// TIA Portal V20 program export: 0 tag tables, 0 data types, 1 data blocks, 3 code blocks (in call order from the OBs), 2 instance data blocks

DATA_BLOCK "MotorSequence_Settings"   // DB2
{ S7_Optimized_Access := 'FALSE' }
VERSION : 1.0
// stored: AutoNumber true, DBAccessibleFromOPCUA true, DBAccessibleFromWebserver true, IsOnlyStoredInLoadMemory false, IsWriteProtectedInAS false
   VAR RETAIN
      StartInterval : Time := T#2S;
      StopInterval : Time := T#2S;
   END_VAR
BEGIN
END_DATA_BLOCK

ORGANIZATION_BLOCK "Main"   // OB1, LAD, ProgramCycle
TITLE = "Main Program Sweep (Cycle)"
{ S7_Optimized_Access := 'TRUE' }
VERSION : 0.1
// stored: AutoNumber false, IsIECCheckEnabled false, SetENOAutomatically false
   VAR_INPUT
      Initial_Call : Bool;
      Remanence : Bool;
   END_VAR
BEGIN

REGION Network 1
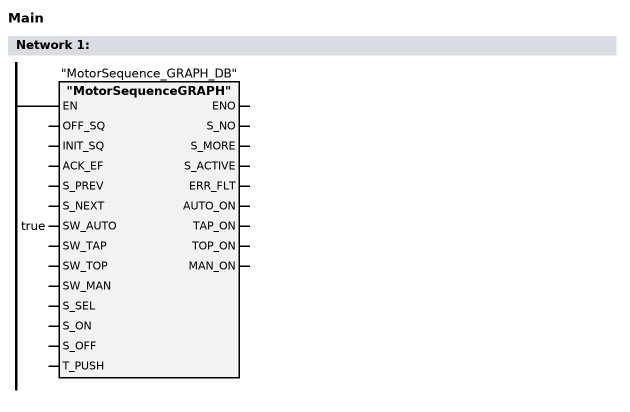
   RUNG wire#powerrail
      "MotorSequence_GRAPH_DB"(SW_AUTO := true, OFF_SQ :=, INIT_SQ :=, ACK_EF :=, S_PREV :=, S_NEXT :=, SW_TAP :=, SW_TOP :=, SW_MAN :=, S_SEL :=, S_ON :=, S_OFF :=, T_PUSH :=, S_NO =>, S_MORE =>, S_ACTIVE =>, ERR_FLT =>, AUTO_ON =>, TAP_ON =>, TOP_ON =>, MAN_ON =>)
   END_RUNG
   // the same network as SCL:
   "MotorSequence_GRAPH_DB"(SW_AUTO := true);   // "MotorSequenceGRAPH"
END_REGION
END_ORGANIZATION_BLOCK

FUNCTION_BLOCK "MotorSequenceGRAPH"   // FB2, GRAPH
VERSION : 0.1
// stored: AcknowledgeErrorsRequired true, AutoNumber false, GraphVersion 6.0, InitialValuesAcquisition false, IsIECCheckEnabled false, LanguageInNetworks LAD, LockOperatingMode false, PermanentILProcessingInMANMode false, SetENOAutomatically false, SkipSteps false, UDAEnableTagReadback false, WithAlarmHandling true
   // inherited from GRAPH_BASE
   VAR
      OFF_SQ_BASE : Bool;
   END_VAR
   VAR_INPUT
      OFF_SQ { ExternalAccessible := 'False'; ExternalVisible := 'False'; ExternalWritable := 'False'} : Bool := false;   // 关闭顺控器
      INIT_SQ { ExternalAccessible := 'False'; ExternalVisible := 'False'; ExternalWritable := 'False'} : Bool := false;   // 将顺序设置为初始状态
      ACK_EF { ExternalAccessible := 'False'; ExternalVisible := 'False'; ExternalWritable := 'False'} : Bool := false;   // 确认所有的错误和故障
      S_PREV { ExternalAccessible := 'False'; ExternalVisible := 'False'; ExternalWritable := 'False'} : Bool := false;   // 在S_NO输出参数中显示前导步
      S_NEXT { ExternalAccessible := 'False'; ExternalVisible := 'False'; ExternalWritable := 'False'} : Bool := false;   // 在S_NO输出参数中显示后续步。
      SW_AUTO { ExternalAccessible := 'False'; ExternalVisible := 'False'; ExternalWritable := 'False'} : Bool := false;   // 自动模式
      SW_TAP { ExternalAccessible := 'False'; ExternalVisible := 'False'; ExternalWritable := 'False'} : Bool := false;   // 半自动/转换条件切换
      SW_TOP { ExternalAccessible := 'False'; ExternalVisible := 'False'; ExternalWritable := 'False'} : Bool := false;   // 半自动/忽略转换条件
      SW_MAN { ExternalAccessible := 'False'; ExternalVisible := 'False'; ExternalWritable := 'False'} : Bool := false;   // 手动模式
      S_SEL { ExternalAccessible := 'False'; ExternalVisible := 'False'; ExternalWritable := 'False'} : Int := 0;   // 选择要在 S_NO中输出的步。
      S_ON { ExternalAccessible := 'False'; ExternalVisible := 'False'; ExternalWritable := 'False'} : Bool := false;   // 激活S_NO 中显示的步。
      S_OFF { ExternalAccessible := 'False'; ExternalVisible := 'False'; ExternalWritable := 'False'} : Bool := false;   // 禁用 S_NO 中标识的步
      T_PUSH { ExternalAccessible := 'False'; ExternalVisible := 'False'; ExternalWritable := 'False'} : Bool := false;   // 允许在半自动模式下跳过转换条件。
   END_VAR
   VAR_OUTPUT
      S_NO { ExternalAccessible := 'False'; ExternalVisible := 'False'; ExternalWritable := 'False'} : Int := 0;   // 步编号
      S_MORE { ExternalAccessible := 'False'; ExternalVisible := 'False'; ExternalWritable := 'False'} : Bool := false;   // 更多步可用，并可在S_NO中显示。
      S_ACTIVE { ExternalAccessible := 'False'; ExternalVisible := 'False'; ExternalWritable := 'False'} : Bool := false;   // 在S_NO 中显示的步是激活的。
      ERR_FLT { ExternalAccessible := 'False'; ExternalVisible := 'False'; ExternalWritable := 'False'} : Bool := false;   // 互锁条件或监控条件组出错
      AUTO_ON { ExternalAccessible := 'False'; ExternalVisible := 'False'; ExternalWritable := 'False'} : Bool := false;   // 当前为自动模式
      TAP_ON { ExternalAccessible := 'False'; ExternalVisible := 'False'; ExternalWritable := 'False'} : Bool := false;   // 已启用SW_TAP模式。
      TOP_ON { ExternalAccessible := 'False'; ExternalVisible := 'False'; ExternalWritable := 'False'} : Bool := false;   // 启用半自动模式/忽略转换条件。
      MAN_ON { ExternalAccessible := 'False'; ExternalVisible := 'False'; ExternalWritable := 'False'} : Bool := false;   // 已启用手动模式。
   END_VAR
BEGIN
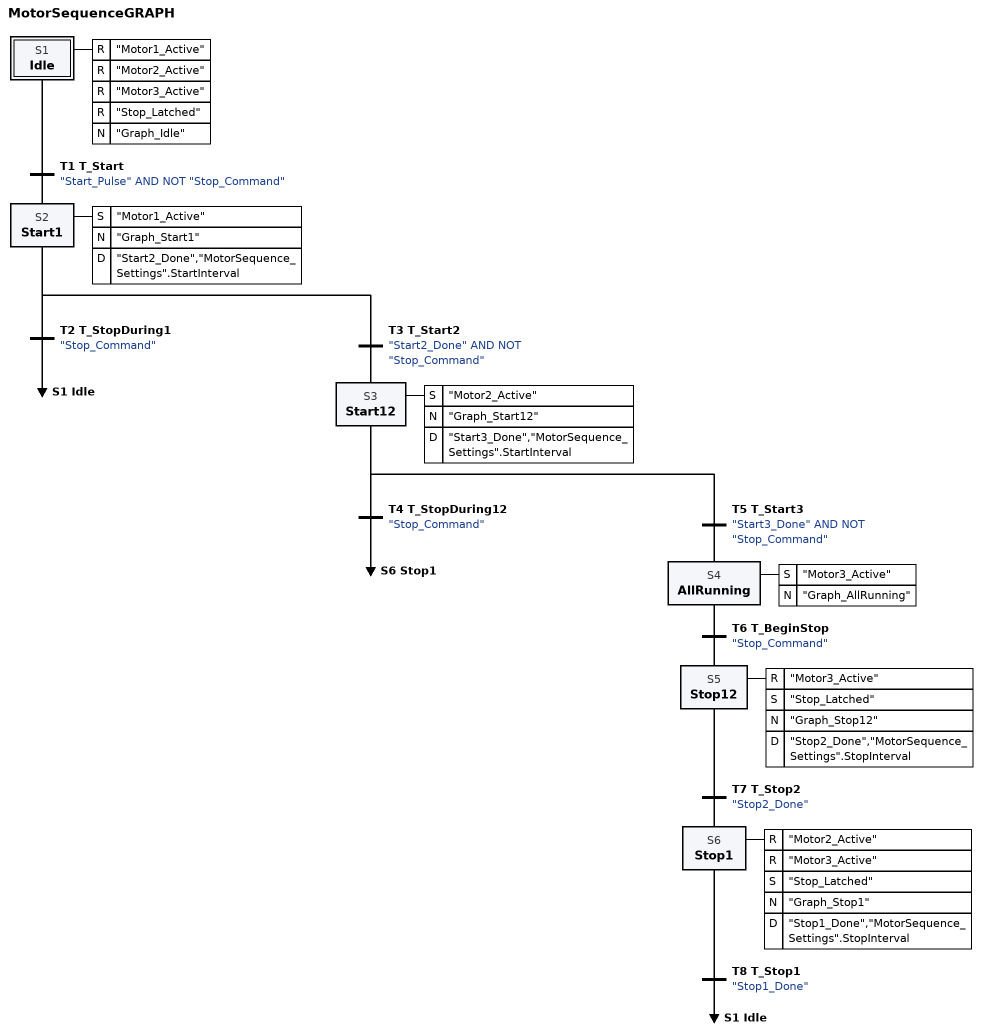
   // permanent pre-instructions
   NETWORK 1
      "Start_Pulse" := "Start_Command" AND NOT "Start_Previous";

   // sequencer 1: 三电机顺序启停：DB2可设间隔
   // 停止优先；停止阶段保持到全部停止；长按启动不自动重启。使用GRAPH原生D延时动作。
   INITIAL_STEP Idle:   // S1, max time T#0ms, warning time T#0ms
      supervision V := "Stop_Command" AND NOT "Stop_Command";
      // 空闲：全部停止，等待新的启动上升沿
              R    "Motor1_Active"
              R    "Motor2_Active"
              R    "Motor3_Active"
              R    "Stop_Latched"
              N    "Graph_Idle"
   END_STEP
   TRANSITION T_Start FROM Idle TO Start1   // T1
      := "Start_Pulse" AND NOT "Stop_Command";
   END_TRANSITION
   STEP Start1:   // S2, max time T#0ms, warning time T#0ms
      supervision V := "Stop_Command" AND NOT "Stop_Command";
      // 1号运行：等待启动间隔，停止优先
              S    "Motor1_Active"
              N    "Graph_Start1"
              D    "Start2_Done","MotorSequence_Settings".StartInterval
   END_STEP
   TRANSITION T_StopDuring1 FROM Start1 TO Idle   // T2, jump
      := "Stop_Command";
   END_TRANSITION
   TRANSITION T_Start2 FROM Start1 TO Start12   // T3
      := "Start2_Done" AND NOT "Stop_Command";
   END_TRANSITION
   STEP Start12:   // S3, max time T#0ms, warning time T#0ms
      supervision V := "Stop_Command" AND NOT "Stop_Command";
      // 1、2号运行：等待启动间隔，停止可跳至只留1号
              S    "Motor2_Active"
              N    "Graph_Start12"
              D    "Start3_Done","MotorSequence_Settings".StartInterval
   END_STEP
   TRANSITION T_StopDuring12 FROM Start12 TO Stop1   // T4, jump
      := "Stop_Command";
   END_TRANSITION
   TRANSITION T_Start3 FROM Start12 TO AllRunning   // T5
      := "Start3_Done" AND NOT "Stop_Command";
   END_TRANSITION
   STEP AllRunning:   // S4, max time T#0ms, warning time T#0ms
      supervision V := "Stop_Command" AND NOT "Stop_Command";
      // 三台电机全部运行，等待停止
              S    "Motor3_Active"
              N    "Graph_AllRunning"
   END_STEP
   TRANSITION T_BeginStop FROM AllRunning TO Stop12   // T6
      := "Stop_Command";
   END_TRANSITION
   STEP Stop12:   // S5, max time T#0ms, warning time T#0ms
      supervision V := "Stop_Command" AND NOT "Stop_Command";
      // 立即停3号，锁存停止序列，等待停止间隔
              R    "Motor3_Active"
              S    "Stop_Latched"
              N    "Graph_Stop12"
              D    "Stop2_Done","MotorSequence_Settings".StopInterval
   END_STEP
   TRANSITION T_Stop2 FROM Stop12 TO Stop1   // T7
      := "Stop2_Done";
   END_TRANSITION
   STEP Stop1:   // S6, max time T#0ms, warning time T#0ms
      supervision V := "Stop_Command" AND NOT "Stop_Command";
      // 立即停2号，保持1号至停止间隔结束
              R    "Motor2_Active"
              R    "Motor3_Active"
              S    "Stop_Latched"
              N    "Graph_Stop1"
              D    "Stop1_Done","MotorSequence_Settings".StopInterval
   END_STEP
   TRANSITION T_Stop1 FROM Stop1 TO Idle   // T8, jump
      := "Stop1_Done";
   END_TRANSITION

   // permanent post-instructions
   NETWORK 1
      "Motor_1" := "Motor1_Active";
   NETWORK 2
      "Motor_2" := "Motor2_Active";
   NETWORK 3
      "Motor_3" := "Motor3_Active";
   NETWORK 4
      "Start_Previous" := "Start_Command";
END_FUNCTION_BLOCK

FUNCTION_BLOCK "MotorSequenceLAD"   // FB1, LAD
{ S7_Optimized_Access := 'TRUE' }
VERSION : 0.1
// stored: AutoNumber true, IsIECCheckEnabled false, IsRetainMemResEnabled false, MemoryReserve 100, SetENOAutomatically false, UDAEnableTagReadback false
   VAR
      Start2 { S7_SetPoint := 'True'} : TON_TIME;
      Start3 { S7_SetPoint := 'True'} : TON_TIME;
      Stop2 { S7_SetPoint := 'True'} : TON_TIME;
      Stop1 { S7_SetPoint := 'True'} : TON_TIME;
   END_VAR
BEGIN

REGION Network 1: 启动上升沿，仅接受新的按钮动作
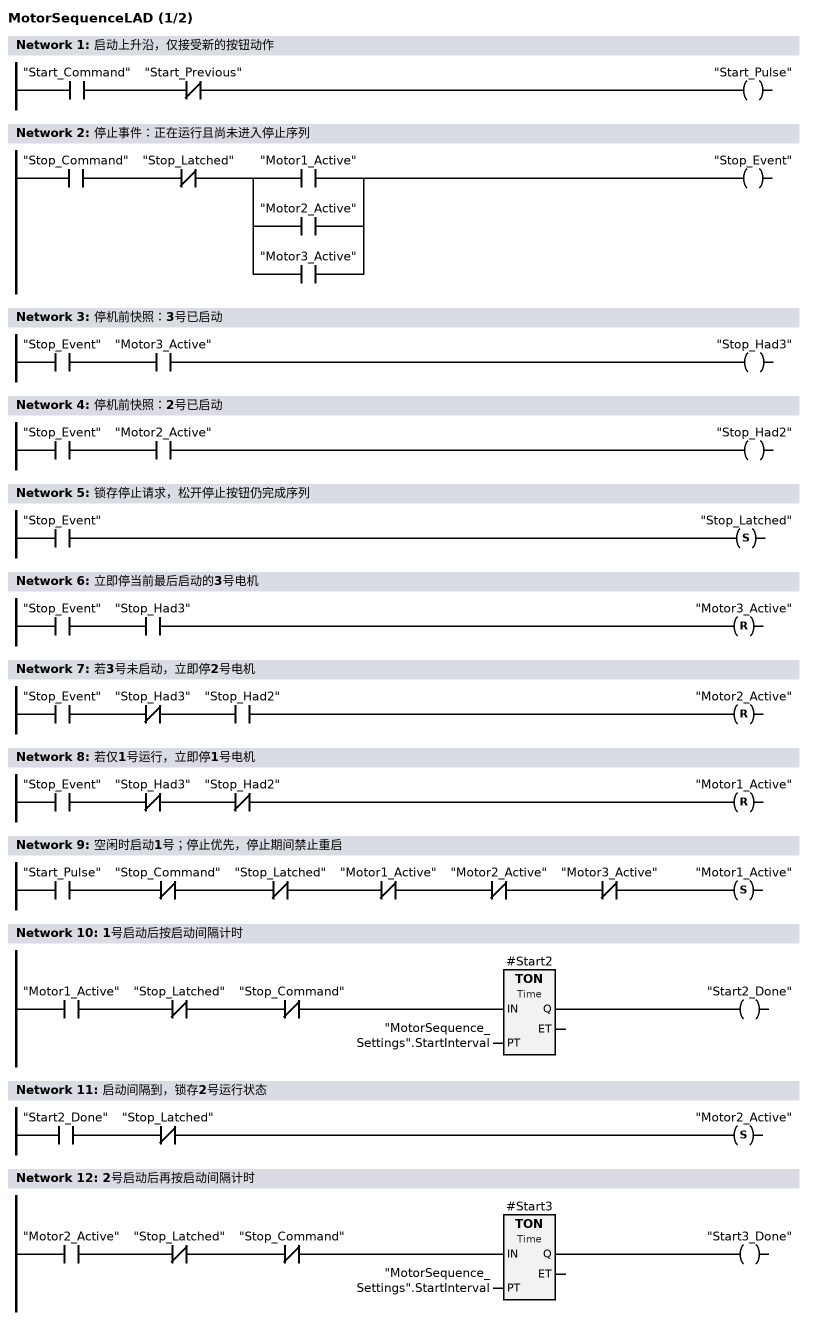
   RUNG wire#powerrail
      Contact( "Start_Command" )
      I_Contact( "Start_Previous" )
      Coil( "Start_Pulse" )
   END_RUNG
   // the same network as SCL:
   "Start_Pulse" := "Start_Command" AND NOT "Start_Previous";
END_REGION

REGION Network 2: 停止事件：正在运行且尚未进入停止序列
   RUNG wire#powerrail
      Contact( "Stop_Command" )
      I_Contact( "Stop_Latched" )
      wire#w1
      Contact( "Motor1_Active" )
      wire#w2
      Coil( "Stop_Event" )
   END_RUNG
   RUNG wire#w1
      Contact( "Motor2_Active" )
   END_RUNG wire#w2
   RUNG wire#w1
      Contact( "Motor3_Active" )
   END_RUNG wire#w2
   // the same network as SCL:
   "Stop_Event" := "Stop_Command" AND NOT "Stop_Latched" AND ("Motor1_Active" OR "Motor2_Active" OR "Motor3_Active");
END_REGION

REGION Network 3: 停机前快照：3号已启动
   RUNG wire#powerrail
      Contact( "Stop_Event" )
      Contact( "Motor3_Active" )
      Coil( "Stop_Had3" )
   END_RUNG
   // the same network as SCL:
   "Stop_Had3" := "Stop_Event" AND "Motor3_Active";
END_REGION

REGION Network 4: 停机前快照：2号已启动
   RUNG wire#powerrail
      Contact( "Stop_Event" )
      Contact( "Motor2_Active" )
      Coil( "Stop_Had2" )
   END_RUNG
   // the same network as SCL:
   "Stop_Had2" := "Stop_Event" AND "Motor2_Active";
END_REGION

REGION Network 5: 锁存停止请求，松开停止按钮仍完成序列
   RUNG wire#powerrail
      Contact( "Stop_Event" )
      S_Coil( "Stop_Latched" )
   END_RUNG
   // the same network as SCL:
   IF "Stop_Event" THEN "Stop_Latched" := TRUE; END_IF;
END_REGION

REGION Network 6: 立即停当前最后启动的3号电机
   RUNG wire#powerrail
      Contact( "Stop_Event" )
      Contact( "Stop_Had3" )
      R_Coil( "Motor3_Active" )
   END_RUNG
   // the same network as SCL:
   IF "Stop_Event" AND "Stop_Had3" THEN "Motor3_Active" := FALSE; END_IF;
END_REGION

REGION Network 7: 若3号未启动，立即停2号电机
   RUNG wire#powerrail
      Contact( "Stop_Event" )
      I_Contact( "Stop_Had3" )
      Contact( "Stop_Had2" )
      R_Coil( "Motor2_Active" )
   END_RUNG
   // the same network as SCL:
   IF "Stop_Event" AND NOT "Stop_Had3" AND "Stop_Had2" THEN "Motor2_Active" := FALSE; END_IF;
END_REGION

REGION Network 8: 若仅1号运行，立即停1号电机
   RUNG wire#powerrail
      Contact( "Stop_Event" )
      I_Contact( "Stop_Had3" )
      I_Contact( "Stop_Had2" )
      R_Coil( "Motor1_Active" )
   END_RUNG
   // the same network as SCL:
   IF "Stop_Event" AND NOT "Stop_Had3" AND NOT "Stop_Had2" THEN "Motor1_Active" := FALSE; END_IF;
END_REGION

REGION Network 9: 空闲时启动1号；停止优先，停止期间禁止重启
   RUNG wire#powerrail
      Contact( "Start_Pulse" )
      I_Contact( "Stop_Command" )
      I_Contact( "Stop_Latched" )
      I_Contact( "Motor1_Active" )
      I_Contact( "Motor2_Active" )
      I_Contact( "Motor3_Active" )
      S_Coil( "Motor1_Active" )
   END_RUNG
   // the same network as SCL:
   IF "Start_Pulse" AND NOT "Stop_Command" AND NOT "Stop_Latched" AND NOT "Motor1_Active" AND NOT "Motor2_Active" AND NOT "Motor3_Active" THEN
       "Motor1_Active" := TRUE;
   END_IF;
END_REGION

REGION Network 10: 1号启动后按启动间隔计时
   RUNG wire#powerrail
      Contact( "Motor1_Active" )
      I_Contact( "Stop_Latched" )
      I_Contact( "Stop_Command" )
      { S7_Templates := "time_type := Time" } #Start2.TON(pt := "MotorSequence_Settings".StartInterval, et =>)
      Coil( "Start2_Done" )
   END_RUNG
   // the same network as SCL:
   #Start2(IN := "Motor1_Active" AND NOT "Stop_Latched" AND NOT "Stop_Command",   // TON
           PT := "MotorSequence_Settings".StartInterval);
   "Start2_Done" := #Start2.Q;
END_REGION

REGION Network 11: 启动间隔到，锁存2号运行状态
   RUNG wire#powerrail
      Contact( "Start2_Done" )
      I_Contact( "Stop_Latched" )
      S_Coil( "Motor2_Active" )
   END_RUNG
   // the same network as SCL:
   IF "Start2_Done" AND NOT "Stop_Latched" THEN "Motor2_Active" := TRUE; END_IF;
END_REGION

REGION Network 12: 2号启动后再按启动间隔计时
   RUNG wire#powerrail
      Contact( "Motor2_Active" )
      I_Contact( "Stop_Latched" )
      I_Contact( "Stop_Command" )
      { S7_Templates := "time_type := Time" } #Start3.TON(pt := "MotorSequence_Settings".StartInterval, et =>)
      Coil( "Start3_Done" )
   END_RUNG
   // the same network as SCL:
   #Start3(IN := "Motor2_Active" AND NOT "Stop_Latched" AND NOT "Stop_Command",   // TON
           PT := "MotorSequence_Settings".StartInterval);
   "Start3_Done" := #Start3.Q;
END_REGION

REGION Network 13: 启动间隔到，锁存3号运行状态
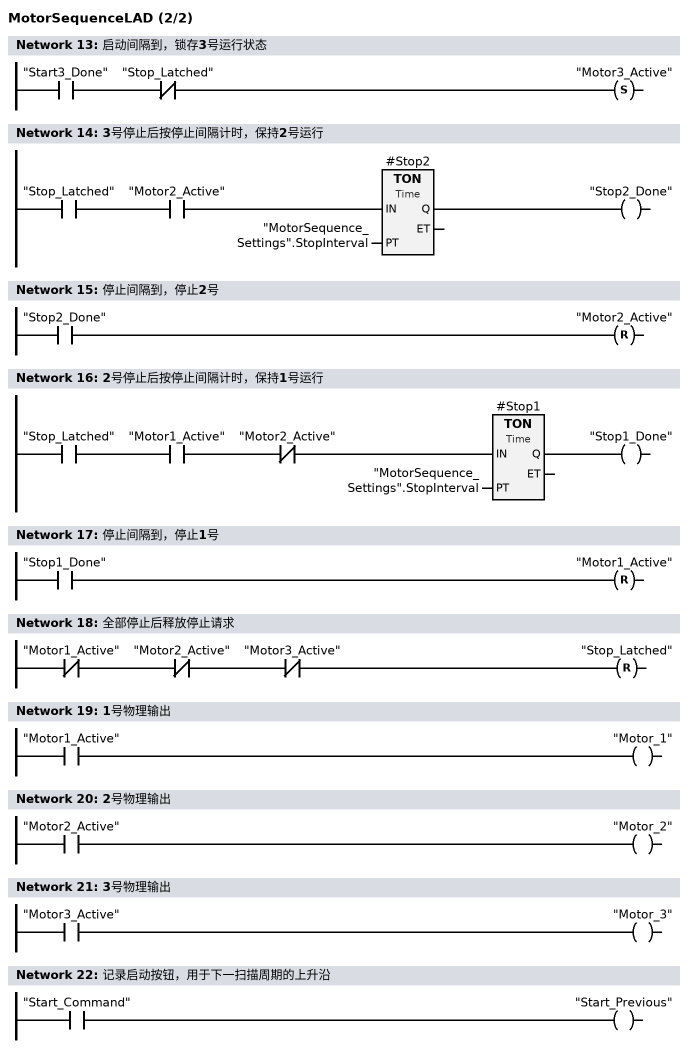
   RUNG wire#powerrail
      Contact( "Start3_Done" )
      I_Contact( "Stop_Latched" )
      S_Coil( "Motor3_Active" )
   END_RUNG
   // the same network as SCL:
   IF "Start3_Done" AND NOT "Stop_Latched" THEN "Motor3_Active" := TRUE; END_IF;
END_REGION

REGION Network 14: 3号停止后按停止间隔计时，保持2号运行
   RUNG wire#powerrail
      Contact( "Stop_Latched" )
      Contact( "Motor2_Active" )
      { S7_Templates := "time_type := Time" } #Stop2.TON(pt := "MotorSequence_Settings".StopInterval, et =>)
      Coil( "Stop2_Done" )
   END_RUNG
   // the same network as SCL:
   #Stop2(IN := "Stop_Latched" AND "Motor2_Active", PT := "MotorSequence_Settings".StopInterval);   // TON
   "Stop2_Done" := #Stop2.Q;
END_REGION

REGION Network 15: 停止间隔到，停止2号
   RUNG wire#powerrail
      Contact( "Stop2_Done" )
      R_Coil( "Motor2_Active" )
   END_RUNG
   // the same network as SCL:
   IF "Stop2_Done" THEN "Motor2_Active" := FALSE; END_IF;
END_REGION

REGION Network 16: 2号停止后按停止间隔计时，保持1号运行
   RUNG wire#powerrail
      Contact( "Stop_Latched" )
      Contact( "Motor1_Active" )
      I_Contact( "Motor2_Active" )
      { S7_Templates := "time_type := Time" } #Stop1.TON(pt := "MotorSequence_Settings".StopInterval, et =>)
      Coil( "Stop1_Done" )
   END_RUNG
   // the same network as SCL:
   #Stop1(IN := "Stop_Latched" AND "Motor1_Active" AND NOT "Motor2_Active",   // TON
          PT := "MotorSequence_Settings".StopInterval);
   "Stop1_Done" := #Stop1.Q;
END_REGION

REGION Network 17: 停止间隔到，停止1号
   RUNG wire#powerrail
      Contact( "Stop1_Done" )
      R_Coil( "Motor1_Active" )
   END_RUNG
   // the same network as SCL:
   IF "Stop1_Done" THEN "Motor1_Active" := FALSE; END_IF;
END_REGION

REGION Network 18: 全部停止后释放停止请求
   RUNG wire#powerrail
      I_Contact( "Motor1_Active" )
      I_Contact( "Motor2_Active" )
      I_Contact( "Motor3_Active" )
      R_Coil( "Stop_Latched" )
   END_RUNG
   // the same network as SCL:
   IF NOT "Motor1_Active" AND NOT "Motor2_Active" AND NOT "Motor3_Active" THEN
       "Stop_Latched" := FALSE;
   END_IF;
END_REGION

REGION Network 19: 1号物理输出
   RUNG wire#powerrail
      Contact( "Motor1_Active" )
      Coil( "Motor_1" )
   END_RUNG
   // the same network as SCL:
   "Motor_1" := "Motor1_Active";
END_REGION

REGION Network 20: 2号物理输出
   RUNG wire#powerrail
      Contact( "Motor2_Active" )
      Coil( "Motor_2" )
   END_RUNG
   // the same network as SCL:
   "Motor_2" := "Motor2_Active";
END_REGION

REGION Network 21: 3号物理输出
   RUNG wire#powerrail
      Contact( "Motor3_Active" )
      Coil( "Motor_3" )
   END_RUNG
   // the same network as SCL:
   "Motor_3" := "Motor3_Active";
END_REGION

REGION Network 22: 记录启动按钮，用于下一扫描周期的上升沿
   RUNG wire#powerrail
      Contact( "Start_Command" )
      Coil( "Start_Previous" )
   END_RUNG
   // the same network as SCL:
   "Start_Previous" := "Start_Command";
END_REGION
END_FUNCTION_BLOCK

DATA_BLOCK "MotorSequence_DB"   // DB1
VERSION : 0.1
// stored: AutoNumber true, DBAccessibleFromOPCUA true, DBAccessibleFromWebserver true, InstanceOfName MotorSequenceLAD, InstanceOfType FB
"MotorSequenceLAD"
BEGIN
END_DATA_BLOCK

DATA_BLOCK "MotorSequence_GRAPH_DB"   // DB3
VERSION : 0.1
// stored: AutoNumber false, DBAccessibleFromOPCUA true, DBAccessibleFromWebserver true, InstanceOfName MotorSequenceGRAPH, InstanceOfType FB
"MotorSequenceGRAPH"
BEGIN
END_DATA_BLOCK
